KUKA KRL program: tipdress1.src, tipdress1.dat

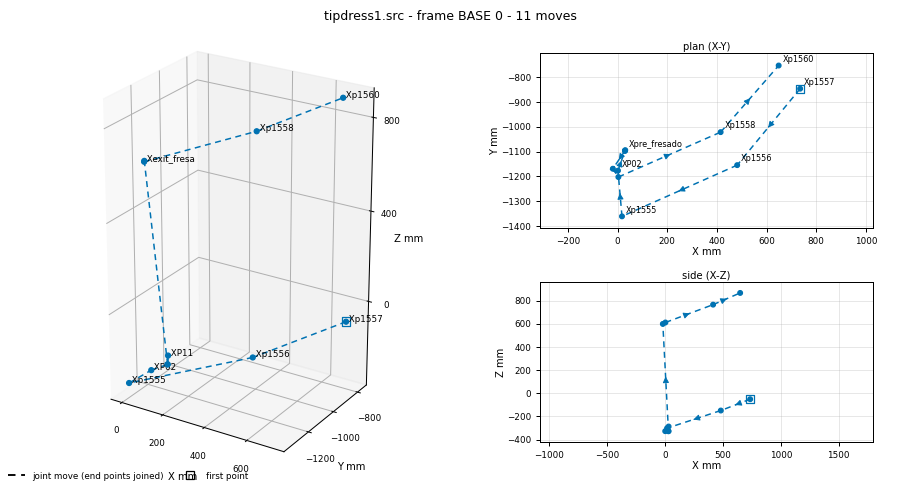
[picture p0: tool path of tipdress1.src in frame BASE 0, 11 of 12 moves have a stored position in this frame; points joined in program order, loops and branches not executed]
--- tipdress1.src ---
&ACCESS RV1
&REL 49
&COMMENT TIPDRESS EXTERNAL GUN 1
DEF tipdress1( )
;================================================
; MODEL    :
; IE GROUP :
; STATION  :
; ROBOT    :
; FUNCTION : TIPDRESS EXTERNAL GUN 1
;================================================
;FOLD INI
;FOLD BASISTECH INI
GLOBAL INTERRUPT DECL 3 WHEN $STOPMESS==TRUE DO IR_STOPM ( )
INTERRUPT ON 3
BAS (#INITMOV,0 )
;ENDFOLD (BASISTECH INI)
;FOLD SPOTTECH INI
USERSPOT(#INIT)
;ENDFOLD (SPOTTECH INI)
;FOLD GRIPPERTECH INI
USER_GRP(0,DUMMY,DUMMY,GDEFAULT)
;ENDFOLD (GRIPPERTECH INI)
;FOLD USER INI
;Make your modifications here
;ENDFOLD (USER INI)
;ENDFOLD (INI)


pgno1_type=0

;FOLD PTP home Vel=100 % H;%{PE}%R 5.6.13,%MKUKATPBASIS,%CMOVE,%VPTP,%P 1:PTP, 2:home, 3:, 5:100, 7:H
$BWDSTART=FALSE
PDAT_ACT=PH
FDAT_ACT=Fhome
BAS(#PTP_PARAMS,100)
$H_POS=XHOME
PTP Xhome
;ENDFOLD
;FOLD PTP p1557 CONT Vel=100 % H Tool[1]:weld Base[0];%{PE}%R 5.6.13,%MKUKATPBASIS,%CMOVE,%VPTP,%P 1:PTP, 2:p1557, 3:C_PTP, 5:100, 7:H
$BWDSTART=FALSE
PDAT_ACT=PH
FDAT_ACT=Fp1557
BAS(#PTP_PARAMS,100)
PTP Xp1557 C_PTP
;ENDFOLD
;FOLD PTP p1556 CONT Vel=100 % H Tool[1]:weld Base[0];%{PE}%R 5.6.13,%MKUKATPBASIS,%CMOVE,%VPTP,%P 1:PTP, 2:p1556, 3:C_PTP, 5:100, 7:H
$BWDSTART=FALSE
PDAT_ACT=PH
FDAT_ACT=Fp1556
BAS(#PTP_PARAMS,100)
PTP Xp1556 C_PTP
;ENDFOLD
;FOLD PTP p1555 CONT Vel=100 % H Tool[1]:weld Base[0];%{PE}%R 5.6.13,%MKUKATPBASIS,%CMOVE,%VPTP,%P 1:PTP, 2:p1555, 3:C_PTP, 5:100, 7:H
$BWDSTART=FALSE
PDAT_ACT=PH
FDAT_ACT=Fp1555
BAS(#PTP_PARAMS,100)
PTP Xp1555 C_PTP
;ENDFOLD
;FOLD PTP P02 CONT Vel=100 % H Tool[1]:weld Base[0];%{PE}%R 5.6.13,%MKUKATPBASIS,%CMOVE,%VPTP,%P 1:PTP, 2:P02, 3:C_PTP, 5:100, 7:H
$BWDSTART=FALSE
PDAT_ACT=PH
FDAT_ACT=FP02
BAS(#PTP_PARAMS,100)
PTP XP02 C_PTP
;ENDFOLD
;FOLD PTP pre_fresado Vel=100 % H Tool[1]:weld Base[0];%{PE}%R 5.6.13,%MKUKATPBASIS,%CMOVE,%VPTP,%P 1:PTP, 2:pre_fresado, 3:, 5:100, 7:H
$BWDSTART=FALSE
PDAT_ACT=PH
FDAT_ACT=Fpre_fresado
BAS(#PTP_PARAMS,100)
PTP Xpre_fresado
;ENDFOLD

REPEAT

;FOLD TDRESS.Select_Active_Electrode 1 ;%{PE}%MKUKATPUSER
B_TDRESS=TDRESS (#TD_SEL ,1)
;ENDFOLD

pgno1_type=0
PGNO1=62

;FOLD TDRESS.Start_Cutter_Gun 1 ;%{PE}%MKUKATPUSER
B_TDRESS=TDRESS (#TD_START ,1)
;ENDFOLD

;FOLD TDRESS.Start_Count_Rotations 1 ;%{PE}%MKUKATPUSER
B_TDRESS=TDRESS (#CNT_STRT ,1)
;ENDFOLD

;FOLD PTP P11 H RETR OPN Gun= 1 Pair= FIRST Tool[1]:weld Base[0];%{PE}%R 6.1.2,%MKUKATPSPOT,%CRETR,%VPTP,%P 1:PTP, 2:P11, 3:, 5:100, 7:H, 9:#OPN, 11:1, 13:#FIRST
$BWDSTART=FALSE
PDAT_ACT=PH
FDAT_ACT=FP11
BAS(#PTP_PARAMS,PH.VEL)
S_ACT.GUN=1
S_ACT.PAIR=#FIRST
S_ACT.RETR=#OPN
S_READY=FALSE
TRIGGER WHEN DISTANCE=1 DELAY=0.0 DO USERSPOT(#RETR, S_ACT) PRIO=-1
PTP XP11
WAIT FOR S_READY

;ENDFOLD

;FOLD CLOSE GUN 1 (3 TIMES) AND CHECK
$ADVANCE=0

FOR I=1 TO  3
CLOSEGUN (1 )

WAIT SEC 0.7



OPENGUN (1 )
ENDFOR
$ADVANCE=3
;endfold

;FOLD PTP pre_fresado Vel=100 % H Tool[1]:weld Base[0];%{PE}%R 5.6.13,%MKUKATPBASIS,%CMOVE,%VPTP,%P 1:PTP, 2:pre_fresado, 3:, 5:100, 7:H
$BWDSTART=FALSE
PDAT_ACT=PH
FDAT_ACT=Fpre_fresado
BAS(#PTP_PARAMS,100)
PTP Xpre_fresado
;ENDFOLD

;FOLD TDRESS.Stop_Count_Rotations 1 ;%{PE}%MKUKATPUSER
B_TDRESS=TDRESS (#CNT_STOP ,1)
;ENDFOLD

;FOLD TDRESS.Check_Rotations_Gun 1 Amount Of Rotations , 2 ;%{PE}%MKUKATPUSER
B_TDRESS=TDRESS (#CNT_CHK ,1, 2)
;ENDFOLD

UNTIL B_TDRESS==TRUE

;FOLD TDRESS.Reset_Counter_Timer 1  Gun nr, 1 ;%{PE}%MKUKATPUSER
B_TDRESS=TDRESS (#TD_RES_CNT ,1, 1)
;ENDFOLD

;FOLD PTP exit_fresa Vel=100 % H Tool[15]:PINZA SOLDADURA Base[0];%{PE}%R 5.6.13,%MKUKATPBASIS,%CMOVE,%VPTP,%P 1:PTP, 2:exit_fresa, 3:, 5:100, 7:H
$BWDSTART=FALSE
PDAT_ACT=PH
FDAT_ACT=Fexit_fresa
BAS(#PTP_PARAMS,100)
PTP Xexit_fresa
;ENDFOLD
;FOLD PTP Best_Praktisch H SPOT Gun= 1 Pair= FIRST RETR OPN INDEX1= 60 INDEX2= 1 Tool[14]:C520 Sin Pieza Base[0];%{PE}%R 6.1.2,%MKUKATPSPOT,%CSPOT,%VPTP,%P 1:PTP, 2:Best_Praktisch, 3:, 5:100, 7:H, 10:1, 12:#FIRST, 14:#OPN, 16:60, 18:1, 20:0, 22:0, 24:0, 25:SDAT3
$BWDSTART=FALSE
PDAT_ACT=PH
FDAT_ACT=FBest_Praktisch
BAS(#PTP_PARAMS,PH.VEL)
S_ACT.GUN=1
S_ACT.PAIR=#FIRST
S_ACT.RETR=#OPN
S_ACT.CLO_TM=SDEFAULT.CLO_TM
S_ACT.PGNO1=60
S_ACT.PGNO2=1
S_ACT.PRESS1=SDEFAULT.PRESS1
S_ACT.PRESS2=SDEFAULT.PRESS2
S_READY=FALSE
USERSPOT(#ADVSPOT, S_ACT)
TRIGGER WHEN DISTANCE=1 DELAY=SDEFAULT.CLO_TM DO USERSPOT(#PRESPOT, S_ACT) PRIO=-1
TRIGGER WHEN DISTANCE=1 DELAY=0.0 DO USERSPOT(#SPOT, S_ACT) PRIO=-1
PTP XBest_Praktisch
WAIT FOR S_READY
;ENDFOLD
;FOLD PTP p1558 CONT Vel=100 % H Tool[15] Base[0];%{PE}%R 5.6.13,%MKUKATPBASIS,%CMOVE,%VPTP,%P 1:PTP, 2:p1558, 3:C_PTP, 5:100, 7:H
$BWDSTART=FALSE
PDAT_ACT=PH
FDAT_ACT=Fp1558
BAS(#PTP_PARAMS,100)
PTP Xp1558 C_PTP
;ENDFOLD
;FOLD PTP p1560 CONT Vel=100 % H Tool[15] Base[0];%{PE}%R 5.6.13,%MKUKATPBASIS,%CMOVE,%VPTP,%P 1:PTP, 2:p1560, 3:C_PTP, 5:100, 7:H
$BWDSTART=FALSE
PDAT_ACT=PH
FDAT_ACT=Fp1560
BAS(#PTP_PARAMS,100)
PTP Xp1560 C_PTP
;ENDFOLD

END

;FOLD SETOUTPUT - SETS OUTPUT IF CONDITIONS ARE OK
DEF  SETOUTPUT (NR :IN,STATE :IN )
;************************************************************
;Function:  sets if to state value
;************************************************************
INT NR
BOOL STATE

IF (NR<>0) THEN
IF (NR>0) THEN
CONTINUE
$OUT[NR]=STATE
ELSE
CONTINUE
$OUT[-NR]= NOT STATE
ENDIF
ENDIF
END ;SetOutput
;ENDFOLD

;FOLD CHKINPUT - CHECKS INPUT <1 & RETURNS INPUT VALUE
DEFFCT  BOOL CHKINPUT(NR :IN,STATE :IN)
;************************************************************
;Function: checks if input nr<1 and returns input value
;************************************************************
INT NR
BOOL STATE

IF (NR<>0) THEN
IF (NR>0) THEN
RETURN  ($IN[NR]==STATE)
ELSE
RETURN  ($IN[-NR]==STATE)
ENDIF
ELSE
RETURN  (TRUE)
ENDIF
ENDFCT ; ChkInput
;ENDFOLD

;FOLD TIMEOUT - WAITS FOR CONDITION WITH TIMEOUT
DEFFCT  BOOL TIMEOUT(CONDITION :OUT,STATE :IN,MAXTIME :IN)
;************************************************************
;Function: waits for condition with timeout
;************************************************************
BOOL CONDITION
BOOL STATE
REAL MAXTIME

$TIMER[5]=-MAXTIME*1000
$TIMER_STOP[5]=FALSE
WHILE  (CONDITION<>STATE) AND  NOT ($TIMER_FLAG[5])
ENDWHILE
RETURN  ($TIMER_FLAG[5])
ENDFCT ; of TimeOut
;ENDFOLD

;FOLD CLOSEGUN - CLOSES WELDGUN BEFORE WELDING
DEF  CLOSEGUN (MYGUN :IN )
;************************************************************
;Function: closes and checks a gun
;************************************************************
INT MYGUN

SETOUTPUT (GRIPPER[MYGUN].OUT2,FALSE )
PULSE ($OUT[GRIPPER[MYGUN].OUT1],TRUE,0.2)
$TIMER[5]=-WAITTIME*1000
$TIMER_STOP[5]=FALSE
WHILE  ((CHKINPUT(GRIPPER[MYGUN].IN1,TRUE) AND CHKINPUT(GRIPPER[MYGUN].IN2,FALSE) AND CHKINPUT(GRIPPER[MYGUN].IN3,FALSE))<>TRUE) AND  NOT ($TIMER_FLAG[5])
ENDWHILE
IF ($TIMER_FLAG[5]) THEN
ERROR_DCP=TRUE
$MSG_T.RELEASE=FALSE
EMPTY_MSG={MSG_T: VALID FALSE,RELEASE FALSE,TYP #NOTIFY,MODUL[] " ",KEY[] " ",PARAM_TYP #VALUE,PARAM[] " ",DLG_FORMAT[] " ",ANSWER 0}
$MSG_T.TYP=#STATE
$MSG_T.KEY[]="Prestroke not closed        "
$MSG_T.VALID=TRUE
WAIT FOR  (($IN[GRIPPER[MYGUN].IN1]==TRUE) AND ($IN[GRIPPER[MYGUN].IN2]==FALSE) AND ($IN[GRIPPER[MYGUN].IN3]==FALSE))
$MSG_T.RELEASE=TRUE
WHILE $MSG_T.VALID
ENDWHILE
ERROR_DCP=FALSE
ENDIF

SETOUTPUT (GRIPPER[MYGUN].OUT3,TRUE )
SETOUTPUT (GRIPPER[MYGUN].OUT4,TRUE )
$TIMER[5]=-WAITTIME*1000
$TIMER_STOP[5]=FALSE
WHILE  ((CHKINPUT(GRIPPER[MYGUN].IN1,FALSE) AND CHKINPUT(GRIPPER[MYGUN].IN2,FALSE) AND CHKINPUT(GRIPPER[MYGUN].IN3,TRUE))<>TRUE) AND  NOT ($TIMER_FLAG[5])
ENDWHILE
IF ($TIMER_FLAG[5]) THEN
ERROR_DCP=TRUE
$MSG_T.RELEASE=FALSE
EMPTY_MSG={MSG_T: VALID FALSE,RELEASE FALSE,TYP #NOTIFY,MODUL[] " ",KEY[] " ",PARAM_TYP #VALUE,PARAM[] " ",DLG_FORMAT[] " ",ANSWER 0}
$MSG_T.TYP=#STATE
$MSG_T.KEY[]="Weldstroke not closed              "
$MSG_T.VALID=TRUE
WAIT FOR  (($IN[GRIPPER[MYGUN].IN1]==FALSE) AND ($IN[GRIPPER[MYGUN].IN2]==FALSE) AND ($IN[GRIPPER[MYGUN].IN3]==TRUE))
$MSG_T.RELEASE=TRUE
WHILE $MSG_T.VALID
ENDWHILE
ERROR_DCP=FALSE
ENDIF

END ;CLOSEGUN

;ENDFOLD

;FOLD OPENGUN - OPENS GUN FULLY AFTER WELDING
DEF  OPENGUN (MYGUN :IN )
;************************************************************
;Function: opens and checks a gun
;************************************************************
INT MYGUN
INT ANSWER

SETOUTPUT (GRIPPER[MYGUN].OUT3,FALSE )
SETOUTPUT (GRIPPER[MYGUN].OUT4,FALSE )
SETOUTPUT (GRIPPER[MYGUN].OUT1,FALSE )
PULSE ($OUT[GRIPPER[MYGUN].OUT2],TRUE,0.2)
$TIMER[5]=-WAITTIME*1000
$TIMER_STOP[5]=FALSE
WHILE  ((CHKINPUT(GRIPPER[MYGUN].IN1,FALSE) AND CHKINPUT(GRIPPER[MYGUN].IN2,TRUE) AND CHKINPUT(GRIPPER[MYGUN].IN3,FALSE))<>TRUE) AND  NOT ($TIMER_FLAG[5])
ENDWHILE
IF ($TIMER_FLAG[5]) THEN
ERROR_DCP=TRUE
$MSG_T.RELEASE=FALSE
EMPTY_MSG={MSG_T: VALID FALSE,RELEASE FALSE,TYP #NOTIFY,MODUL[] " ",KEY[] " ",PARAM_TYP #VALUE,PARAM[] " ",DLG_FORMAT[] " ",ANSWER 0}
$MSG_T.TYP=#STATE
$MSG_T.KEY[]="Prestroke not open                 "
$MSG_T.VALID=TRUE
WAIT FOR  (($IN[GRIPPER[MYGUN].IN1]==FALSE) AND ($IN[GRIPPER[MYGUN].IN2]==TRUE) AND ($IN[GRIPPER[MYGUN].IN3]==FALSE))
$MSG_T.RELEASE=TRUE
WHILE $MSG_T.VALID
ENDWHILE
ERROR_DCP=FALSE
ENDIF

END ;OPENGUN

--- tipdress1.dat ---
&ACCESS RV1
&REL 49
&COMMENT TIPDRESS EXTERNAL GUN 1
DEFDAT  TIPDRESS1
;FOLD EXTERNAL DECLARATIONS;%{PE}%MKUKATPBASIS,%CEXT,%VCOMMON,%P
;FOLD GRIPPERTECH EXT
EXT  H50 (INT  :IN,INT  :IN,INT  :IN,GRP_TYP  :IN )
;ENDFOLD (GRIPPERTECH EXT)
;FOLD SPOTTECH EXT
EXT  USERSPOT (S_COMMAND  :IN,SPOT_TYPE  :IN )
;ENDFOLD (SPOTTECH EXT)
;FOLD BASISTECH EXT;%{PE}%MKUKATPBASIS,%CEXT,%VEXT,%P
EXT  BAS (BAS_COMMAND  :IN,REAL  :IN )
DECL INT SUCCESS
;ENDFOLD (BASISTECH EXT)
;FOLD USER EXT;%{E}%MKUKATPUSER,%CEXT,%VEXT,%P
;Make here your modifications
;ENDFOLD (USER EXT)
;ENDFOLD (EXTERNAL DECLERATIONS)
;FOLD USER EXT;%{}%V2.2.2,%MKUKATPUSER,%CEXT,%VEXT,%P
;Make here your modifications
DECL BOOL TIPKONTROLE
DECL INT ANSWER
DECL INT WAITTIME=5
;ENDFOLD
;ENDFOLD
DECL INT I

;******************************
;*     E6POS Declarations     *
;******************************

DECL E6POS XP10={X 30.7658501,Y -1094.01099,Z -286.682404,A 25.4987392,B 1.97903597,C -0.329104304,S 6,T 26,E1 0.0,E2 0.0,E3 0.0,E4 0.0,E5 0.0,E6 0.0}
DECL E6POS XP20={X -1662.00305,Y -1200.49304,Z 238.679993,A 92.3594437,B 77.6989288,C -175.853195,S 6,T 26,E1 -667.745789,E2 0.0,E3 0.0,E4 0.0,E5 0.0,E6 0.0}
DECL E6POS XBEFORETIPDRESS={X -1664.84497,Y -1195.28101,Z 131.821106,A 92.7083206,B 79.2879791,C -177.241806,S 6,T 26,E1 -667.74939,E2 0.0,E3 0.0,E4 0.0,E5 0.0,E6 0.0}
DECL E6POS XDRESS_POS={X -1664.83301,Y -1250.33301,Z 131.817993,A 92.7068863,B 79.2882233,C -177.243393,S 6,T 26,E1 -667.74762,E2 0.0,E3 0.0,E4 0.0,E5 0.0,E6 0.0}
DECL E6POS XAFTERTIPDRESS={X -1664.84497,Y -1195.28101,Z 131.821106,A 92.7083206,B 79.2879791,C -177.241806,S 6,T 26,E1 -667.74939,E2 0.0,E3 0.0,E4 0.0,E5 0.0,E6 0.0}
DECL E6POS XBEST_PRACKTICE={X -1662.02905,Y -1184.83496,Z 277.771301,A 92.3578873,B 77.6946869,C -175.853302,S 6,T 26,E1 -667.74762,E2 0.0,E3 0.0,E4 0.0,E5 0.0,E6 0.0}
DECL E6POS XP30={X -958.122009,Y 929.273499,Z 985.610474,A 92.0788727,B 72.5539932,C -179.8358,S 6,T 26,E1 -2887.17505,E2 0.0,E3 0.0,E4 0.0,E5 0.0,E6 0.0}

;******************************
;*      FDAT Declarations     *
;******************************

DECL FDAT FP10={TOOL_NO 1,BASE_NO 0,IPO_FRAME #BASE,TQ_STATE FALSE}
DECL FDAT FP20={TOOL_NO 1,BASE_NO 0,IPO_FRAME #BASE}
DECL FDAT FBEFORETIPDRESS={TOOL_NO 1,BASE_NO 0,IPO_FRAME #BASE}
DECL FDAT FDRESS_POS={TOOL_NO 1,BASE_NO 0,IPO_FRAME #BASE}
DECL FDAT FAFTERTIPDRESS={TOOL_NO 1,BASE_NO 0,IPO_FRAME #BASE}
DECL FDAT FBEST_PRACKTICE={TOOL_NO 1,BASE_NO 0,IPO_FRAME #BASE}
DECL FDAT FP30={TOOL_NO 1,BASE_NO 0,IPO_FRAME #BASE}

;******************************
;*  PDAT & LDAT Declarations  *
;******************************

DECL PDAT PH={VEL 100.0,ACC 100.0,APO_DIST 100.0,APO_MODE #CPTP}

DECL E6POS XBEST_PRAKTISCH={X 3.06066203,Y -1202.17297,Z 611.93042,A -125.567596,B -7.38407087,C -173.644897,S 6,T 26,E1 0.0,E2 0.0,E3 0.0,E4 0.0,E5 0.0,E6 0.0}
DECL SPOT_SUGG_T LAST_SPOT={GUN[] "1                       ",RETR_CMD[] "#OPN                    ",CHOISE[] "#FIRST                  ",CLO_TM[] "0                       ",PGNO1[] "1                       ",PRESS1[] "0                       ",PGNO2[] "1                       ",PRESS2[] "0                       ",SPOT_PARAMS[] "SDAT3                   "}
DECL BASIS_SUGG_T LAST_BASIS={POINT1[] "p1560                   ",POINT2[] "p1560                   ",CP_PARAMS[] "CPDAT0                  ",PTP_PARAMS[] "H                       ",CONT[] "C_PTP                   ",CP_VEL[] "2.0                     ",PTP_VEL[] "100                     ",SYNC_PARAMS[] "SYNCDAT                 ",SPL_NAME[] "S0                      "}
DECL FDAT FBest_Praktisch={TOOL_NO 14,BASE_NO 0,IPO_FRAME #BASE,POINT2[] " ",TQ_STATE FALSE}
DECL PDAT PPDAT1={VEL 100.0,ACC 100.0,APO_DIST 100.0}
DECL E6POS XBest_Praktice={X -1662.07202,Y -1184.76196,Z 277.795013,A 92.3631592,B 77.6921463,C -175.8461,S 6,T 26,E1 -667.74762,E2 0.0,E3 0.0,E4 0.0,E5 0.0,E6 0.0}
DECL FDAT FBest_Praktice={TOOL_NO 1,BASE_NO 0,IPO_FRAME #BASE,POINT2[] " "}
DECL E6POS XP21={X -929.55603,Y -159.533905,Z 748.283386,A 92.0804672,B 72.5703812,C -179.830597,S 6,T 26,E1 -2646.86792,E2 0.0,E3 0.0,E4 0.0,E5 0.0,E6 0.0}
DECL FDAT FP21={TOOL_NO 1,BASE_NO 0,IPO_FRAME #BASE}
DECL E6POS XP31={X -1185.09497,Y -662.41571,Z 415.422485,A 99.845192,B 75.8905869,C -168.599792,S 6,T 26,E1 -1294.38501,E2 0.0,E3 0.0,E4 0.0,E5 0.0,E6 0.0}
DECL FDAT FP31={TOOL_NO 1,BASE_NO 0,IPO_FRAME #BASE}
DECL E6POS XP01={X -521.268372,Y 932.237488,Z 809.362427,A -104.869499,B 25.3531094,C 156.8172,S 2,T 43,E1 0.0,E2 0.0,E3 0.0,E4 0.0,E5 0.0,E6 0.0}
DECL FDAT FP01={TOOL_NO 15,BASE_NO 0,IPO_FRAME #BASE,POINT2[] " ",TQ_STATE FALSE}
DECL E6POS XP02={X 1.47015905,Y -1176.46594,Z -326.900909,A 24.0927391,B 2.20976591,C -0.817254126,S 6,T 26,E1 0.0,E2 0.0,E3 0.0,E4 0.0,E5 0.0,E6 0.0}
DECL FDAT FP02={TOOL_NO 1,BASE_NO 0,IPO_FRAME #BASE,POINT2[] " ",TQ_STATE FALSE}
DECL E6POS XP022={X -545.304504,Y 780.863586,Z 303.431,A -96.6869965,B -0.146422103,C 179.108505,S 2,T 43,E1 0.0,E2 0.0,E3 0.0,E4 0.0,E5 0.0,E6 0.0}
DECL FDAT FP022={TOOL_NO 15,BASE_NO 0,IPO_FRAME #BASE,POINT2[] " ",TQ_STATE FALSE}
DECL E6POS XEXIT_FRESA={X -19.1423302,Y -1168.72705,Z 599.551025,A -125.410202,B 0.478198886,C -178.771393,S 6,T 26,E1 0.0,E2 0.0,E3 0.0,E4 0.0,E5 0.0,E6 0.0}
DECL FDAT Fexit_fresa={TOOL_NO 15,BASE_NO 0,IPO_FRAME #BASE,POINT2[] " ",TQ_STATE FALSE}
DECL E6POS XEXIT_FRESA_2={X -521.27002,Y 932.235901,Z 809.362793,A -104.869301,B 25.3530197,C 156.8172,S 2,T 43,E1 0.0,E2 0.0,E3 0.0,E4 0.0,E5 0.0,E6 0.0}
DECL FDAT Fexit_fresa_2={TOOL_NO 15,BASE_NO 0,IPO_FRAME #BASE,POINT2[] " ",TQ_STATE FALSE}
DECL E6POS XPRE_FRESADO={X 29.4938698,Y -1096.56396,Z -327.138885,A 25.4940891,B 1.89127803,C -0.142933503,S 6,T 26,E1 0.0,E2 0.0,E3 0.0,E4 0.0,E5 0.0,E6 0.0}
DECL FDAT Fpre_fresado={TOOL_NO 1,BASE_NO 0,IPO_FRAME #BASE,POINT2[] " ",TQ_STATE FALSE}
DECL E6POS XP1555={X 17.5958195,Y -1360.61597,Z -301.022308,A 23.6130409,B 6.36468601,C -9.25088882,S 6,T 26,E1 0.0,E2 0.0,E3 0.0,E4 0.0,E5 0.0,E6 0.0}
DECL FDAT Fp1555={TOOL_NO 1,BASE_NO 0,IPO_FRAME #BASE,POINT2[] " ",TQ_STATE FALSE}
DECL E6POS XP1556={X 481.643494,Y -1154.31702,Z -148.6595,A 30.6545601,B 3.87480402,C -9.08418941,S 6,T 26,E1 0.0,E2 0.0,E3 0.0,E4 0.0,E5 0.0,E6 0.0}
DECL FDAT Fp1556={TOOL_NO 1,BASE_NO 0,IPO_FRAME #BASE,POINT2[] " ",TQ_STATE FALSE}
DECL E6POS XP1557={X 735.259827,Y -846.376282,Z -50.7595787,A 36.4931488,B 2.33025098,C -7.71590185,S 6,T 26,E1 0.0,E2 0.0,E3 0.0,E4 0.0,E5 0.0,E6 0.0}
DECL FDAT Fp1557={TOOL_NO 1,BASE_NO 0,IPO_FRAME #BASE,POINT2[] " ",TQ_STATE FALSE}
DECL E6POS XP1558={X 415.015991,Y -1021.36499,Z 766.043091,A -118.665298,B -5.1592021,C -172.507797,S 6,T 26,E1 0.0,E2 0.0,E3 0.0,E4 0.0,E5 0.0,E6 0.0}
DECL FDAT Fp1558={TOOL_NO 15,BASE_NO 0,IPO_FRAME #BASE,POINT2[] " ",TQ_STATE FALSE}
DECL E6POS XP1559={X 648.731079,Y -753.047424,Z 867.173096,A -112.872597,B -3.13396502,C -172.896606,S 6,T 26,E1 0.0,E2 0.0,E3 0.0,E4 0.0,E5 0.0,E6 0.0}
DECL FDAT Fp1559={TOOL_NO 15,BASE_NO 0,IPO_FRAME #BASE,POINT2[] " ",TQ_STATE FALSE}
DECL E6POS XP1560={X 648.731079,Y -753.047424,Z 867.173096,A -112.872597,B -3.13396502,C -172.896606,S 6,T 26,E1 0.0,E2 0.0,E3 0.0,E4 0.0,E5 0.0,E6 0.0}
DECL FDAT Fp1560={TOOL_NO 15,BASE_NO 0,IPO_FRAME #BASE,POINT2[] " ",TQ_STATE FALSE}
DECL E6POS XP11={X 30.7658501,Y -1094.01099,Z -286.682404,A 25.4987392,B 1.97903597,C -0.329104304,S 6,T 26,E1 0.0,E2 0.0,E3 0.0,E4 0.0,E5 0.0,E6 0.0}
DECL FDAT FP11={TOOL_NO 1,BASE_NO 0,IPO_FRAME #BASE,TQ_STATE FALSE}
ENDDAT
